FUNCTION_BLOCK FB_FlowTransform
VAR_INPUT
	bEnable : BOOL;
	nRawInput : INT;
END_VAR
VAR_OUTPUT
	fOutput : LREAL;
	fOutputBit : LREAL;
END_VAR
VAR
	fRawInput : LREAL;
	fTempInput : LREAL;
	fTempOutput : LREAL;
	fMaxInputValue			: LREAL := 32767.0;
	fNeutralInputValue  	: LREAL := 15250.0;
	fMinInputValue 			: LREAL := 0.0;
	
	fNeutralDeadband		: LREAL := 25.0;
	
	fMaxOutputValue  		: LREAL := 150.0;
	fNeutralOutputValue  	: LREAL := 0.0;
	fMinOutputValue  		: LREAL := -150.0;
	
END_VAR

fRawInput := INT_TO_LREAL(nRawInput);

fTempInput := fRawInput - fNeutralInputValue;

IF fTempInput > fNeutralDeadband THEN
	fTempOutput := fMaxOutputValue * fTempInput/(fMaxInputValue - fNeutralInputValue);
ELSIF fTempInput < -fNeutralDeadband THEN	
	fTempOutput := fMinOutputValue * (fTempInput)/(fNeutralInputValue - fMinInputValue);
ELSE
	fTempOutput := 0.0;
END_IF

IF NOT(bEnable) THEN
	fOutput := 0.0;
ELSE
	fOutput := LIMIT(fMinOutputValue, fTempOutput, fMaxOutputValue);
END_IF

fOutputBit := INT_TO_LREAL(nRawInput);

END_FUNCTION_BLOCK

(* stored: Version 1.1.0.1, ProductVersion 3.1.4026.11
   POU FB_FlowTransform: Id {cf40c1a8-0fc0-4809-bdf6-f129a497ed41}, SpecialFunc None *)
